Omron CX-Programmer project NewProject (CX-Programmer 9.61)

# PLC NewPLC1: CP1H X

## Global symbols (name address type ; comment)
D3000.01 BOOL  ; ok

## Program NewProgram1 (cyclic task 0)
Local symbols
P_On CF113 BOOL
p_on BOOL

### Section Section1

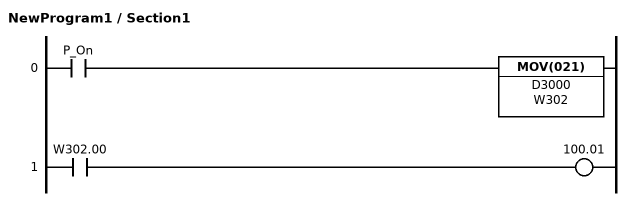
; rung 0
LD P_On
MOV(021) D3000 W302
; rung 1
LD W302.00
OUT 100.01

### Section END
; rung 0
END(001)